ABB RAPID module: MainModule.mod

MODULE MainModule
	CONST robtarget Target_10:=[[291.23,-42.20,675.34],[0.726174,0.418599,0.37568,0.395362],[-1,0,0,1],[9E+09,9E+09,9E+09,9E+09,9E+09,9E+09]];
	CONST robtarget Target_20:=[[364.353866871,131.99897178,359.648693238],[0.353552801,0.612372796,0.612372742,0.353552826],[0,0,0,1],[9E+09,9E+09,9E+09,9E+09,9E+09,9E+09]];
	CONST robtarget Target_30:=[[265.54,-8.35,795.20],[0.758267,0.252794,0.326487,0.504511],[-1,0,0,1],[9E+09,9E+09,9E+09,9E+09,9E+09,9E+09]];
	PROC main()
	    MoveL Target_10,v100,z100,tool0\WObj:=wobj0;
	    MoveL Target_20, v500, z100, tool0\WObj:=wobj0;
	    Stop;
	ENDPROC
ENDMODULE
